// TIA Portal project "Clase 3 SCL" (V14)

(* hardware
DEVICE "S7-1200 station_1"  S7-1200 Station
   slot 0: "Rack_0"  S7-1200 Rack  Rack  V1.0
   slot 1: "PLC_1"  CPU 1214C DC/DC/DC  6ES7 214-1AG40-0XB0  V4.2
*)

// ===== PLC "PLC_1"  CPU 1214C DC/DC/DC =====

VAR_GLOBAL   // PLC tag table "Salidas"
   "Motor (KM1)" AT %Q0.0 : Bool;
END_VAR

VAR_GLOBAL   // PLC tag table "Entradas"
   "Rele termico" AT %I0.0 : Bool;
   "Pulsador Start" AT %I0.1 : Bool;
   "Pulsador Stop" AT %I0.2 : Bool;
   "Seta Emergencia" AT %I0.3 : Bool;
END_VAR

DATA_BLOCK "var"   // DB1
{ S7_Optimized_Access := 'TRUE' }
VERSION : 0.1
   VAR
      General : Struct
         "Sistema OK" : Bool;
         "Act. Motor (KM1)" : Bool;
         Estado : WString;
      END_STRUCT;
      "Contador Pulsos" : Struct
         Reset : Bool;
         Contador : IEC_COUNTER;
      END_STRUCT;
   END_VAR
BEGIN
   "Contador Pulsos".Contador.PV := 6;
END_DATA_BLOCK

FUNCTION "Salidas" : Void   // FC1, SCL
{ S7_Optimized_Access := 'TRUE' }
VERSION : 0.1
BEGIN
   // ACTIVACION DE SALIDAS FISICAS DEL AUTOMATA

   // SALIDA Q0.0
   "Motor (KM1)" := "var".General."Act. Motor (KM1)";
END_FUNCTION

ORGANIZATION_BLOCK "Main"   // OB1, SCL, ProgramCycle
TITLE = "Main Program Sweep (Cycle)"
{ S7_Optimized_Access := 'TRUE' }
VERSION : 0.1
   VAR_INPUT
      Initial_Call : Bool;   // Initial call of this OB
      Remanence : Bool;   // =True, if remanent data are available
   END_VAR
BEGIN
   // PROGRAMA MAIN DE CONTADOR DE PULSOS

   // Llamamos al bloque FC1
   "Salidas"();

   Region Estructura de programa
       Region Condicional de seguridad
           "var".General."Sistema OK" := "Rele termico" AND "Seta Emergencia";
       END_REGION
       Region Contador de pulsos
           "var"."Contador Pulsos".Contador.CTU(CU:="var".General."Sistema OK" AND "Pulsador Start",
                                                R:="var"."Contador Pulsos".Reset OR NOT "var".General."Sistema OK" OR NOT "Pulsador Stop",
                                                PV:="var"."Contador Pulsos".Contador.PV,
                                                Q=>"var"."Contador Pulsos".Reset,
                                                CV=>"var"."Contador Pulsos".Contador.CV);
       END_REGION
       Region Condicional funcionamiento motor
           If "var"."Contador Pulsos".Contador.CV = 4 THEN
               "var".General."Act. Motor (KM1)" := true;
           ELSIF
               NOT "var".General."Sistema OK" OR NOT "Pulsador Stop" THEN
               "var".General."Act. Motor (KM1)" := false;
           END_IF;
       END_REGION
       Region Instrucción Case
           Case "var"."Contador Pulsos".Contador.CV OF

               0..2:
                   "var".General.Estado := WSTRING#'Estado Inactivo';
               3:
                   "var".General.Estado := WSTRING#'Estado 1';
               4:
                   "var".General.Estado := WSTRING#'Estado Activo';

               ELSE
                   "var".General.Estado := WSTRING#'Alarma';
           END_CASE;
       END_REGION
   END_REGION
END_ORGANIZATION_BLOCK